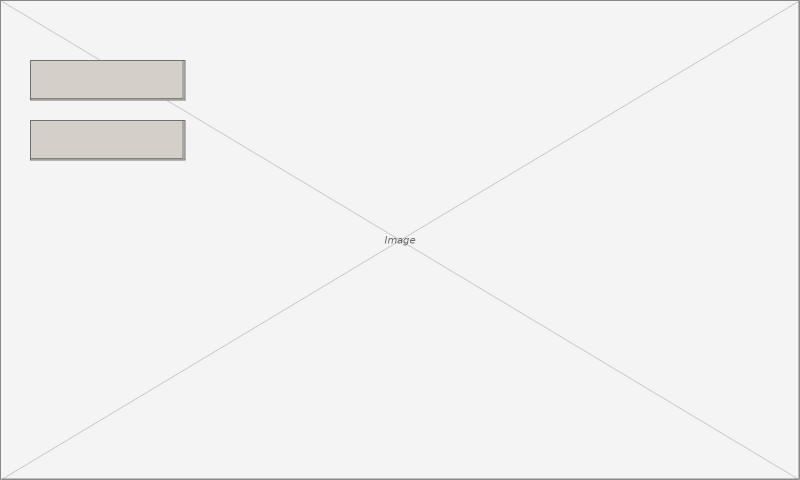
VISUALIZATION autoMode  // 800x480
    Image (0,0 800x480)
        p84334746: MAIN.bmpID
    Button (30,60 155x40), image: Buttons.homeButton
        OnMouseDown: change screen: Main
        OnMouseDown: execute { MAIN.autoModeON:=FALSE; }
    Button (30,120 155x40), image: Buttons.startButton
        OnMouseDown: toggle MAIN.autoModeON
END_VISUALIZATION

(* stored: Version 1.1.0.1, ProductVersion 3.1.4018.2
   Visu autoMode: Id {cdb25d90-ad8a-4086-ac38-f26ce2e78d05} *)
